//==================================================================================================
//								RJM Maszyny sp. z o.o.
//									04.02.2022
//	Obsługa elektrozaworu 5/2 nonostabilny
// 	v1.0	|| TC v 3.1.4024.22		|| - pierwsza wersja
//==================================================================================================
FUNCTION_BLOCK FB_Elektrozawor_5na2_1Cewka IMPLEMENTS I_Elektrozawor_5na
VAR
	fbCewka									: FB_ElektrozaworCewka;
END_VAR

//==================================================================================================
//								RJM Maszyny sp. z o.o.
//									04.02.2022
//	Włączenie cewki - wyjscie 2
// 	v1.0	|| TC v 3.1.4024.22		|| - pierwsza wersja
//==================================================================================================
METHOD WlaczWyjscie2 : BOOL
VAR_INPUT
END_VAR
fbCewka.Wylacz ();
END_METHOD

//==================================================================================================
//								RJM Maszyny sp. z o.o.
//									04.02.2022
//	Włączenie cewki - wyjscie 4
// 	v1.0	|| TC v 3.1.4024.22		|| - pierwsza wersja
//==================================================================================================
METHOD WlaczWyjscie4 : BOOL
VAR_INPUT
END_VAR
fbCewka.Wlacz ();
END_METHOD

//==================================================================================================
//								RJM Maszyny sp. z o.o.
//									04.02.2022
//	Wyłączenie cewki - wyjscie 2
// 	v1.0	|| TC v 3.1.4024.22		|| - pierwsza wersja
//==================================================================================================
METHOD WylaczWyjscie2 : BOOL
VAR_INPUT
END_VAR
fbCewka.Wlacz ();
END_METHOD

//==================================================================================================
//								RJM Maszyny sp. z o.o.
//									04.02.2022
//	Wyłączenie cewki - wyjscie 4
// 	v1.0	|| TC v 3.1.4024.22		|| - pierwsza wersja
//==================================================================================================
METHOD WylaczWyjscie4 : BOOL
VAR_INPUT
END_VAR
fbCewka.Wlacz ();
END_METHOD

END_FUNCTION_BLOCK

(* stored: Version 1.1.0.1, ProductVersion 3.1.4024.11
   POU FB_Elektrozawor_5na2_1Cewka: Id {8b33e655-5369-4414-be57-0a6015bb253a}, SpecialFunc None
   Method WlaczWyjscie2: Id {0d3396d8-bc87-4f8a-ad75-eb2b4f532754}
   Method WlaczWyjscie4: Id {5339f3a7-5c31-4d52-a830-356d60810e60}
   Method WylaczWyjscie2: Id {56c7b0f9-5450-44fe-8c4b-6e9773f5fb1e}
   Method WylaczWyjscie4: Id {9f5b7b82-08fc-4311-9921-406c91d3be2f} *)
